// TIA Portal V17 export
// export: Created 2025-03-10T12:18:47.9580326Z, ExportSetting WithDefaults, DisplayName Totally Integrated Automation Portal, DisplayVersion V17 Update 8, DisplayName TIA Portal Openness, DisplayVersion V17 Update 8, DisplayName TIA Portal Version Control Interface, DisplayVersion V17, DisplayName SINAMICS Startdrive Advanced, DisplayVersion V17 SP2, DisplayName SINAMICS Startdrive G110M, G120, G120C, G120D, G120P, G115D, DisplayVersion V17 SP2, DisplayName SINAMICS Startdrive G130, G150, S120, S150, SINAMICS MV, S210, DisplayVersion V17 SP2, DisplayName STEP 7 Professional, DisplayVersion V17 Update 8, DisplayName SINUMERIK ONE STEP 7 Toolbox, DisplayVersion V17 Update 12, DisplayName SINUMERIK 840D sl STEP 7 Toolbox, DisplayVersion V17 Update 12, DisplayName STEP 7 Safety, DisplayVersion V17 Update 6, DisplayName WinCC Advanced, DisplayVersion V17 Update 8
DATA_BLOCK "DB21021_PF_1_HEATER_JKL_UNIT_02"   // DB21021
{ DB_Accessible_From_OPC_UA := 'FALSE' }
VERSION : 0.1
// stored: AutoNumber false, DBAccessibleFromOPCUA false, DBAccessibleFromWebserver true, InstanceOfName FB21012_POWDER_FEEDER_HEATER_JKT, InstanceOfType FB
"FB21012_POWDER_FEEDER_HEATER_JKT"
   // VAR_INPUT
   //    iPF_HEAT_AVAILABLE_OPTION : Bool;
   //    iPF_PROFINET_MODE_ACTIVE_FAULT : Bool;
   //    iPF_HOPPER_TEMP_GrHH_LINE_1 : Bool;
   //    iPF_HOPPER_TEMP_GrHH_LINE_2 : Bool;
   //    iCONTROL_ON_DELAYED : Bool;
   //    iAUTO_START_REQUEST : Bool;
   //    iAUTO_STOP_REQUEST : Bool;
   //    iUNIT_NUMBER : Byte;
   //    iMANUAL_START_REQ_LINE_1 : Bool;
   //    iMANUAL_START_REQ_LINE_2 : Bool;
   //    iMANUAL_STOP_REQ_LINE_1 : Bool;
   //    iMANUAL_STOP_REQ_LINE_2 : Bool;
   // END_VAR
   // VAR_OUTPUT
   //    oPF_HEATING_ON_CMD_LINE_1 : Bool;
   //    oPF_HEATING_ON_CMD_LINE_2 : Bool;
   //    oPF_HEATING_OFF_CMD_LINE_1 : Bool;
   //    oPF_HEATING_OFF_CMD_LINE_2 : Bool;
   //    oSWITCHONCONDITION_ON_LINE_1 : Bool;
   //    oSWITCHONCONDITION_ON_LINE_2 : Bool;
   //    oSWITCHONCONDITION_OFF_LINE_1 : Bool;
   //    oSWITCHONCONDITION_OFF_LINE_2 : Bool;
   //    oMOTION_ACTIVE_RIGHT_LINE_1 : Bool;
   //    oMOTION_ACTIVE_RIGHT_LINE_2 : Bool;
   //    oMOTION_ACTIVE_LEFT_LINE_1 : Bool;
   //    oMOTION_ACTIVE_LEFT_LINE_2 : Bool;
   //    oLIMIT_RIGHT_LINE_1 : Bool;
   //    oLIMIT_RIGHT_LINE_2 : Bool;
   //    oLIMIT_LEFT_LINE_1 : Bool;
   //    oLIMIT_LEFT_LINE_2 : Bool;
   //    oALARM_HOPPER_LINE_1_TEMP_ABOVE_HIGH_LIMIT : Bool;
   //    oALARM_HOPPER_LINE_2_TEMP_ABOVE_HIGH_LIMIT : Bool;
   // END_VAR
   // VAR
   //    DATA : "POWDER FEEDER HEATER JKT";
   //    INPUT_SETTINGS : Struct
   //       UNIT_NUMBER : Int;
   //       FEEDER_NUMBER : Int;
   //    END_STRUCT;
   //    HEATER_STATUS_LINE_1 { S7_SetPoint := 'True'} : Byte;
   //    HEATER_STATUS_LINE_2 : Byte;
   // END_VAR
BEGIN
END_DATA_BLOCK
